FUNCTION_BLOCK ABSTRACT FB_AbstructFuture IMPLEMENTS InterfaceFuture
VAR_INPUT
END_VAR
VAR_OUTPUT
END_VAR
VAR
	{attribute 'TcEncoding':='UTF-8'}
	_future_name :STRING := 'NO_NAME';
	_busy : BOOL; 
	_state : E_FutureExecutionState;
END_VAR

METHOD abort : BOOL // Return TRUE if finish.
abort := TRUE;
END_METHOD

METHOD execute : BOOL // Return TRUE if finish.
END_METHOD

PROPERTY future_name : STRING // Name of future.
GET
future_name := _future_name;
END_GET
SET
_future_name := future_name;
END_SET
END_PROPERTY

METHOD init : BOOL // Return TRUE if finish.
init := TRUE;
END_METHOD

PROPERTY nErrorID : UDINT // Set result code when finished any method. 0 should be set when normal case.
GET
END_GET
END_PROPERTY

METHOD quit : BOOL // Return TRUE if finish.
init();
quit := TRUE;
END_METHOD

{warning 'add property implementation'}
PROPERTY state : E_FutureExecutionState // Execution state of this future.
GET
state := _state;
END_GET
SET
_state := state;
END_SET
END_PROPERTY

END_FUNCTION_BLOCK

(* stored: Version 1.1.0.1, ProductVersion 3.1.4024.12
   POU FB_AbstructFuture: Id {e0e3f6dd-6f71-426e-8a03-d727df6ff260}, SpecialFunc None
   Method abort: Id {862be836-a2ae-4f1d-92dd-4b23d30b26d7}
   Method execute: Id {ba07fa30-bd40-4f42-b8d8-9c368f5519ee}
   Property future_name: Id {2365611b-3978-40e5-af7c-084e8898106e}
   Get Get: Id {e0946a55-87b0-493c-91f5-c6fd2898618e}
   Set Set: Id {16c10530-d9ba-4ec9-9835-68bda488cc9e}
   Method init: Id {0f9a7fa1-ec74-4313-8d46-6183b844e43b}
   Property nErrorID: Id {5e96776e-2ecf-4a2b-b5d9-c234f6343ca2}
   Get Get: Id {60455303-60d8-490d-880a-ad439ea813d7}
   Method quit: Id {0f34e09c-f5ef-4bf1-a724-c006af3b609d}
   Property state: Id {91bd7ebd-9da1-475e-8562-21de65a90ef0}
   Get Get: Id {5f907f7b-f09a-4df2-813b-0a4f8e85b687}
   Set Set: Id {1e6ea7bf-ae29-4091-a681-57ef0260a8f7} *)
